// TIA Portal V18 export
// export: Created 2026-06-11T12:00:00Z, ExportSetting WithDefaults, DisplayName Totally Integrated Automation Portal, DisplayVersion V18, DisplayName TIA Portal Openness, DisplayVersion V18
TagTable "HMI_Tags"
  1400_FT115_PV : Real  (PLC tag 1400_FT115_PV, HMI_Connection_1, 1 s)   // Lưu lượng dòng liệu đo được tại FT115
  1400_FT101_PV : Real  (PLC tag 1400_FT101_PV, HMI_Connection_1, 1 s)   // Lưu lượng dòng liệu đo được tại FT101
  1400_1_02_PV : Real  (PLC tag 1400_1_02_PV, HMI_Connection_1, 1 s)   // Giá trị đo của cảm biến 1-02
  1406_TX35_PV : Real  (PLC tag 1406_TX35_PV, HMI_Connection_1, 1 s)   // Giá trị đo cảm biến nhiệt độ/áp suất TX35
  1400_TT64_PV : Real  (PLC tag 1400_TT64_PV, HMI_Connection_1, 1 s)   // Nhiệt độ đo được tại TT64
  1400_TT32_PV : Real  (PLC tag 1400_TT32_PV, HMI_Connection_1, 1 s)   // Nhiệt độ đo được tại TT32
  1400_LGFE01_PV : Real  (PLC tag 1400_LGFE01_PV, HMI_Connection_1, 1 s)   // Mức bồn hoặc lưu lượng đo tại LGFE01
  1400_FS51_PV : Real  (PLC tag 1400_FS51_PV, HMI_Connection_1, 1 s)   // Giá trị lưu lượng đo được tại FS51
  1400_FY301_PV : Real  (PLC tag 1400_FY301_PV, HMI_Connection_1, 1 s)   // Mức cân hoặc vị trí điều khiển bồn FY301
  1400_TT101_PV : Real  (PLC tag 1400_TT101_PV, HMI_Connection_1, 1 s)   // Nhiệt độ đo được tại TT101
  1400_FTT02_PV : Real  (PLC tag 1400_FTT02_PV, HMI_Connection_1, 1 s)   // Lưu lượng/nhiệt độ đo được tại FTT02
  1500S_Trang_Thai : Bool  (PLC tag 1500S_Trang_Thai, HMI_Connection_1, 1 s)   // Trạng thái hoạt động dòng liệu 1500S (0: Không chảy, 1: Đang chảy)
  1404T_Trang_Thai : Bool  (PLC tag 1404T_Trang_Thai, HMI_Connection_1, 1 s)   // Trạng thái hoạt động dòng liệu 1404T
  CR_2013_FO_104_Trang_Thai : Bool  (PLC tag CR_2013_FO_104_Trang_Thai, HMI_Connection_1, 1 s)   // Trạng thái hoạt động dòng liệu CR-2013-FO-104
  BFOC_SS_20_06_Trang_Thai : Bool  (PLC tag BFOC_SS_20_06_Trang_Thai, HMI_Connection_1, 1 s)   // Trạng thái hoạt động dòng liệu BFOC-SS-20-06
  PC03010T01_Trang_Thai : Bool  (PLC tag PC03010T01_Trang_Thai, HMI_Connection_1, 1 s)   // Trạng thái dòng liệu đầu ra PC03010T01
  1401_Trang_Thai : Bool  (PLC tag 1401_Trang_Thai, HMI_Connection_1, 1 s)   // Trạng thái dòng liệu xả đáy 1401
  1400_PT91_Chay : Bool  (PLC tag 1400_PT91_Chay, HMI_Connection_1, 1 s)   // Tín hiệu báo chạy bơm 1400PT91 (1: Chạy)
  1400_KCK01_Chay : Bool  (PLC tag 1400_KCK01_Chay, HMI_Connection_1, 1 s)   // Tín hiệu báo chạy cánh khuấy bồn 1400KCK01
  1400_FT102_Mo : Bool  (PLC tag 1400_FT102_Mo, HMI_Connection_1, 1 s)   // Tín hiệu báo mở van nạp liệu 1400FT102
  1400_TY33_Mo : Bool  (PLC tag 1400_TY33_Mo, HMI_Connection_1, 1 s)   // Tín hiệu báo mở van điều khiển cooling 1400TY33
  160_FEC53_Mo : Bool  (PLC tag 160_FEC53_Mo, HMI_Connection_1, 1 s)   // Tín hiệu báo mở van kẹp 160 FEC53
  1400_TXC32_Mo : Bool  (PLC tag 1400_TXC32_Mo, HMI_Connection_1, 1 s)   // Tín hiệu báo mở van điều khiển 1400TXC32
  1400_TC32_Mo : Bool  (PLC tag 1400_TC32_Mo, HMI_Connection_1, 1 s)   // Tín hiệu báo mở van điều khiển 1400TC32
  1400_FIC01_Mo : Bool  (PLC tag 1400_FIC01_Mo, HMI_Connection_1, 1 s)   // Tín hiệu báo mở van điều khiển 1400FIC01
  1400_FS51_Mo : Bool  (PLC tag 1400_FS51_Mo, HMI_Connection_1, 1 s)   // Tín hiệu báo mở van xả đáy 1400FS51
  1500S_Status : Int  (PLC tag 1500S_Status, HMI_Connection_1, 1 s)   // Mã trạng thái dòng liệu 1500S (0: Dừng, 1: Chạy, 2: Lỗi)
  1404T_Status : Int  (PLC tag 1404T_Status, HMI_Connection_1, 1 s)   // Mã trạng thái dòng liệu 1404T
  CR_2013_FO_104_Status : Int  (PLC tag CR_2013_FO_104_Status, HMI_Connection_1, 1 s)   // Mã trạng thái dòng liệu CR-2013-FO-104
  BFOC_SS_20_06_Status : Int  (PLC tag BFOC_SS_20_06_Status, HMI_Connection_1, 1 s)   // Mã trạng thái dòng liệu BFOC-SS-20-06
  PC03010T01_Status : Int  (PLC tag PC03010T01_Status, HMI_Connection_1, 1 s)   // Mã trạng thái dòng liệu PC03010T01
  1401_Status : Int  (PLC tag 1401_Status, HMI_Connection_1, 1 s)   // Mã trạng thái dòng liệu xả đáy 1401
  1400_PT91_Status : Int  (PLC tag 1400_PT91_Status, HMI_Connection_1, 1 s)   // Mã trạng thái hoạt động bơm 1400PT91 (0: Dừng, 1: Chạy, 2: Lỗi)
  1400_KCK01_Status : Int  (PLC tag 1400_KCK01_Status, HMI_Connection_1, 1 s)   // Mã trạng thái hoạt động cánh khuấy 1400KCK01
  1400_FT102_Status : Int  (PLC tag 1400_FT102_Status, HMI_Connection_1, 1 s)   // Mã trạng thái hoạt động van 1400FT102 (0: Đóng, 1: Mở, 2: Lỗi)
  1400_TY33_Status : Int  (PLC tag 1400_TY33_Status, HMI_Connection_1, 1 s)   // Mã trạng thái hoạt động van 1400TY33
  160_FEC53_Status : Int  (PLC tag 160_FEC53_Status, HMI_Connection_1, 1 s)   // Mã trạng thái hoạt động van 160 FEC53
  1400_TXC32_Status : Int  (PLC tag 1400_TXC32_Status, HMI_Connection_1, 1 s)   // Mã trạng thái hoạt động van 1400TXC32
  1400_TC32_Status : Int  (PLC tag 1400_TC32_Status, HMI_Connection_1, 1 s)   // Mã trạng thái hoạt động van 1400TC32
  1400_FIC01_Status : Int  (PLC tag 1400_FIC01_Status, HMI_Connection_1, 1 s)   // Mã trạng thái hoạt động van 1400FIC01
  1400_FS51_Status : Int  (PLC tag 1400_FS51_Status, HMI_Connection_1, 1 s)   // Mã trạng thái hoạt động van 1400FS51
